# EPICS substitutions: iocBoot/ioc4idHHLM/substitutions/canberra_3.substitutions
file "$(MCA)/mcaApp/Db/simple_mca.db"
{
pattern
{P           M       DTYP           INP              PREC  CHANS}
{4idHHLM:med:   mca1  "asynMCA"       "@asyn(AIM1/1 0)"  3     2048}
{4idHHLM:med:   mca2  "asynMCA"       "@asyn(AIM1/2 0)"  3     2048}
{4idHHLM:med:   mca3  "asynMCA"       "@asyn(AIM2/1 0)"  3     2048}
{4idHHLM:med:   mca0  "Soft Channel"  ""                 3     2048}
}

#file "$(MCA)/mcaApp/Db/icb_amp.db"
#{
#pattern
#{P			AMP		PORT}
#{4idHHLM:med:	amp1	icbAmp1}
#}

file "$(MCA)/mcaApp/Db/icb_adc.db"
{
pattern
{P			ADC		PORT}
{4idHHLM:med:	adc1	"icbAdc1"}
{4idHHLM:med:	adc2	"icbAdc2"}
{4idHHLM:med:	adc3	"icbAdc3"}
}

#file "$(MCA)/mcaApp/Db/icb_hvps.db"
#{
#pattern
#{P			HVPS	LIMIT	PORT}
#{4idHHLM:med:	hvps1	1000	"icbHvps1"}
#}

file "$(MCA)/mcaApp/Db/icb_tca.db"
{
pattern
{P,          TCA,	PORT,		MCA}
{4idHHLM:med:,  tca1,	"icbTca1",	mca1}
{4idHHLM:med:,  tca2,	"icbTca2",	mca2}
{4idHHLM:med:,  tca3,	"icbTca3",	mca3}
}
